(* IEC 61131-3 sources: LLM-CodeGen-TestGen/Tests/DEC_TO_HEX_2, 2 files *)

(* ---- DEC_TO_HEX_FullTest.st ---- *)
FUNCTION BIT_OF_DWORD : BOOL
  VAR_INPUT
    IN : DWORD;
    N : INT;
  END_VAR

  BIT_OF_DWORD := (SHR(in,N) AND 16#00000001) > 0;
  (* from OSCAT library; www.oscat.de  *)
END_FUNCTION

FUNCTION SIGN_R : BOOL
  VAR_INPUT
    IN : REAL;
  END_VAR

  SIGN_R := in < 0.0;
  (* from OSCAT library; www.oscat.de  *)
END_FUNCTION

FUNCTION FLOOR : INT
  VAR_INPUT
    x : REAL;
  END_VAR

  FLOOR := REAL_TO_INT(X);
  IF INT_TO_REAL(FLOOR) > X THEN
  	floor := floor - 1;
  END_IF;
  (* from OSCAT library; www.oscat.de  *)
END_FUNCTION

FUNCTION FLOOR2 : DINT
  VAR_INPUT
    x : REAL;
  END_VAR

  FLOOR2 := REAL_TO_DINT(X);
  IF DINT_TO_REAL(FLOOR2) > X THEN
  	FLOOR2 := FLOOR2 - DINT#1;
  END_IF;
  (* from OSCAT library; www.oscat.de  *)
END_FUNCTION

FUNCTION MODR : REAL
  VAR_INPUT
    IN : REAL;
    DIVI : REAL;
  END_VAR

  IF divi = 0.0 THEN
  	MODR := 0.0;
  ELSE
  	MODR := in - DINT_TO_REAL(FLOOR2(in / divi)) * divi;
  END_IF;
  (* from OSCAT library; www.oscat.de  *)
  (* FC FLOOR2 required *)
END_FUNCTION

FUNCTION REVERSE : BYTE
  VAR_INPUT
    IN : BYTE;
  END_VAR

  reverse := SHL(in,7) OR SHR(in,7) OR (ROR(in,3) AND BYTE#2#01000100) OR (ROL(in,3) AND BYTE#2#00100010)
  	OR (SHL(in,1) AND BYTE#2#00010000) OR (SHR(in,1) AND BYTE#2#00001000);

  (* Fromm Oscat Library, www.oscat.de *)
END_FUNCTION

FUNCTION REFLECT : DWORD
  VAR_INPUT
    DI : DWORD;
    L : INT;
  END_VAR
  VAR
    i : INT;
    _d : DWORD;
  END_VAR

  _d := DI;
  FOR i := 1 TO L DO
  	REFLECT := SHL(REFLECT, 1) OR BOOL_TO_DWORD((_d AND DWORD#2#0000_0001) > DWORD#0); (* D.0 *)
  	_d := SHR(_d, 1);
  END_FOR;
  REFLECT := REFLECT OR SHL(_d, L);

  (* Fromm Oscat Library, www.oscat.de *)
END_FUNCTION

FUNCTION BIT_LOAD_B : BYTE
  VAR_INPUT
    IN : BYTE;
    VAL : BOOL;
    POS : INT;
  END_VAR

  IF VAL THEN
  	BIT_LOAD_B := in OR SHL(BYTE#1,pos);
  ELSE
  	BIT_LOAD_B := in AND (NOT SHL(BYTE#1,pos));
  END_IF;

  (*From OSCAT Library, www.oscat.de*)
END_FUNCTION

FUNCTION _BYTE_TO_INT : INT
  VAR_INPUT
    IN : BYTE;
  END_VAR

  _BYTE_TO_INT := USINT_TO_INT(BYTE_TO_USINT(IN));

  (*From OSCAT Library, www.oscat.de*)
END_FUNCTION

FUNCTION T_PLC_MS : UDINT
  VAR
    tx : UDINT;
  END_VAR
  VAR_INPUT
    debug : BOOL;
  END_VAR
  VAR
    N : INT := 0;
    offset : UDINT := 0;
    temp : DWORD := 1;
  END_VAR

  tx := 0;
  {extern unsigned long __tick;
  extern unsigned long long common_ticktime__;
  unsigned long long ticktime_ms = (common_ticktime__)/1000000;
  UDINT plc_time = (UDINT)(ticktime_ms * (unsigned long long)__tick);
  TX = plc_time}
  T_PLC_MS := tx;
  IF debug THEN
  	T_PLC_MS := (DWORD_TO_UDINT(SHL(UDINT_TO_DWORD(T_PLC_MS),N) OR SHL(temp,N))-1) + OFFSET;
  END_IF;

  IF debug THEN
  	T_PLC_MS := (DWORD_TO_UDINT(SHL(UDINT_TO_DWORD(T_PLC_MS),N) OR SHL(temp,N))-1) + OFFSET;
  END_IF;

  (* Original Code:
  tx := TIME();
  T_PLC_MS := TIME_TO_DWORD(Tx);
  IF debug THEN
  	T_PLC_MS := (SHL(T_PLC_MS,N) OR SHL(DWORD#1,N)-1) + OFFSET;
  END_IF;
  *)

  (* From OSCAT library, www.oscat.de

  this is a temporary T_PLC_MS FB until OpenPLC gets it´s own time() functionality *)

  (* PLC_TIME and Global variables PLC_SCAN_CYCL and PLC_CYCL_TIME required *)
END_FUNCTION

FUNCTION T_PLC_US : UDINT
  VAR
    tx : UDINT;
  END_VAR
  VAR_INPUT
    debug : BOOL;
  END_VAR
  VAR
    N : INT := 0;
    offset : UDINT := 0;
    temp : DWORD := 1;
  END_VAR

  T_PLC_US := tx*1000;
  IF debug THEN
  	T_PLC_US := (DWORD_TO_UDINT(SHL(UDINT_TO_DWORD(T_PLC_US),N) OR SHL(temp,N))-1) + OFFSET;
  END_IF;

  (* Original Code:
  tx := TIME();
  T_PLC_US := TIME_TO_DWORD(Tx)*1000;
  IF debug THEN
  	T_PLC_US := (SHL(T_PLC_US,N) OR SHL(DWORD#1,N)-1) + OFFSET;
  END_IF;
  *)

  (* From OSCAT library, www.oscat.de

  this is a temporary T_PLC_US FB until OpenPLC gets it´s own time() functionality *)

  (* PLC_TIME and Global variables PLC_SCAN_CYCL and PLC_CYCL_TIME required *)
END_FUNCTION

FUNCTION_BLOCK FT_DERIV
  VAR_INPUT
    IN : REAL;
    K : REAL := 1.0;
    RUN : BOOL := TRUE;
  END_VAR
  VAR_OUTPUT
    OUT : REAL;
  END_VAR
  VAR
    old : REAL;
    tx : UDINT;
    last : UDINT;
    init : BOOL;
    tc : REAL;
  END_VAR

  tx:= T_PLC_US(en:=true);
  tc := UDINT_TO_REAL(tx - last);

  (* init on firsat startup *)
  IF NOT init THEN
  	init := TRUE;
  	old := in;
  ELSIF run AND tc > 0.0 THEN
  	out := (in - old) / tc * 1000000.0 * K;
  	old := in;
  ELSE
  	out := 0.0;
  END_IF;

  last := tx;

  (* From OSCAT Library, www.oscat.de *)
  (* T_PLC_US, required *)
END_FUNCTION_BLOCK

FUNCTION_BLOCK FT_PIWL
  VAR_INPUT
    IN : REAL;
    KP : REAL := 1.0;
    KI : REAL := 1.0;
    LIM_L : REAL := -1.0E38;
    LIM_H : REAL := 1.0E38;
    RST : BOOL;
  END_VAR
  VAR_OUTPUT
    Y : REAL;
    LIM : BOOL;
  END_VAR
  VAR
    init : BOOL;
    tx : UDINT;
    tc : REAL;
    t_last : UDINT;
    in_last : REAL;
    i : REAL;
    p : REAL;
  END_VAR

  IF NOT init OR RST THEN
  	init := TRUE;
  	in_last := in;
  		t_last := T_PLC_US(en:=true);
  	i := 0.0;
  	tc := 0.0;
  ELSE
  	(* read last cycle time in Microseconds *)
  		tx := T_PLC_US(en:=true);
  	tc := UDINT_TO_REAL(tx - t_last);
  	t_last := tx;

  	(* calculate proportional part *)
  	p := KP * IN;

  	(* run integrator *)
  	i := (IN + in_last) * 5.0E-7 * KI * tc + i;
  	in_last := IN;

  	(* calculate output Y *)
  	Y := p + i;

  	(* check output for limits *)
  	IF Y >= LIM_H THEN
  		Y := LIM_H;
  		IF ki <> 0.0 THEN
  			i := LIM_H - p;
  		ELSE
  			i := 0.0;
  		END_IF;
  		LIM := TRUE;
  	ELSIF Y <= LIM_L THEN
  		Y := LIM_L;
  		IF ki <> 0.0 THEN
  			i := LIM_L - p;
  		ELSE
  			i := 0.0;
  		END_IF;
  		LIM := TRUE;
  	ELSE
  		LIM := FALSE;
  	END_IF;
  END_IF;

  (* From OSCAT Library, www.oscat.de *)
  (* T_PLC_US required *)
END_FUNCTION_BLOCK

FUNCTION_BLOCK INTEGRATE
  VAR_INPUT
    _E : BOOL := TRUE;
    X : REAL;
    K : REAL := 1.0;
  END_VAR
  VAR_IN_OUT
    Y : REAL;
  END_VAR
  VAR
    x_last : REAL;
    init : BOOL;
    last : UDINT;
    tx : UDINT;
  END_VAR

  tx:= T_PLC_MS(en:=true);

  IF NOT init THEN
  	init := TRUE;
  	X_last := X;
  ELSIF _E THEN
  	Y := (X + X_LAST) * 0.5E-3 * UDINT_TO_REAL(tx-last) * K + Y;
  	X_last := X;
  END_IF;
  last := tx;

  (* From OSCAT Library, www.oscat.de *)
  (* T_PLC_MS required *)
END_FUNCTION_BLOCK

FUNCTION_BLOCK DEC_TO_HEX
  VAR_INPUT
    DecimalValue : DINT;
  END_VAR
  VAR_OUTPUT
    HexString : STRING;
  END_VAR
  VAR
    i : INT;
    hexDigits : ARRAY [0..15] OF STRING := ['0', '1', '2', '3', '4', '5', '6', '7', '8', '9', 'A', 'B', 'C', 'D', 'E', 'F'];
    digitIndex : INT;
    hexDigit : STRING;
    significantDigitFound : BOOL := FALSE;
    digitValue : DINT;
    powerOfInteger : DINT;
  END_VAR

  HexString := '';

  IF DecimalValue = 0 THEN
      HexString := '0';
      RETURN;
  END_IF;

  significantDigitFound := FALSE;

  FOR digitIndex := 0 TO 7 DO

      powerOfInteger:=1;
      FOR i := 1 TO 7 - digitIndex DO
        powerOfInteger := powerOfInteger * 16;
      END_FOR;

      digitValue := DIV(DecimalValue, powerOfInteger) MOD 16;
      hexDigit := hexDigits[digitValue];

      IF hexDigit <> '0' OR significantDigitFound OR (7 - digitIndex) = 0 THEN
          significantDigitFound := TRUE;
          HexString := CONCAT(HexString, hexDigit);
      END_IF;

  END_FOR;
END_FUNCTION_BLOCK

FUNCTION_BLOCK FB_TEST_0
  VAR_OUTPUT
    Finished : BOOL;
    Failed : BOOL;
  END_VAR
  VAR
    TestBlock : DEC_TO_HEX;
    TestState : INT;
    Timer : TON;
  END_VAR

  Timer(IN:=TRUE, PT:= T#0s); (* placeholder for later usage *)

  CASE testState OF
    0:
      IF (Timer.Q) THEN
        TestBlock(DecimalValue := 0);
        TestState:=TestState+1;
      END_IF;
      Timer(IN:=TRUE, PT:=T#0s);
    1:
      IF (Timer.Q) THEN
      {printf("0,0: TestBlock.HexString = '0'  actual=%s\n", (char*)&__GET_VAR(data__->TESTBLOCK.HEXSTRING,).body);}
        IF NOT(TestBlock.HexString = '0') THEN Failed := TRUE; END_IF;
      END_IF;
      Finished:=TRUE;
  END_CASE;
END_FUNCTION_BLOCK

FUNCTION_BLOCK FB_TEST_1
  VAR_OUTPUT
    Finished : BOOL;
    Failed : BOOL;
  END_VAR
  VAR
    TestBlock : DEC_TO_HEX;
    TestState : INT;
    Timer : TON;
  END_VAR

  Timer(IN:=TRUE, PT:= T#0s); (* placeholder for later usage *)

  CASE testState OF
    0:
      IF (Timer.Q) THEN
        TestBlock(DecimalValue := 1);
        TestState:=TestState+1;
      END_IF;
      Timer(IN:=TRUE, PT:=T#0s);
    1:
      IF (Timer.Q) THEN
      {printf("1,0: TestBlock.HexString = '1'  actual=%s\n", (char*)&__GET_VAR(data__->TESTBLOCK.HEXSTRING,).body);}
        IF NOT(TestBlock.HexString = '1') THEN Failed := TRUE; END_IF;
      END_IF;
      Finished:=TRUE;
  END_CASE;
END_FUNCTION_BLOCK

FUNCTION_BLOCK FB_TEST_2
  VAR_OUTPUT
    Finished : BOOL;
    Failed : BOOL;
  END_VAR
  VAR
    TestBlock : DEC_TO_HEX;
    TestState : INT;
    Timer : TON;
  END_VAR

  Timer(IN:=TRUE, PT:= T#0s); (* placeholder for later usage *)

  CASE testState OF
    0:
      IF (Timer.Q) THEN
        TestBlock(DecimalValue := 10);
        TestState:=TestState+1;
      END_IF;
      Timer(IN:=TRUE, PT:=T#0s);
    1:
      IF (Timer.Q) THEN
      {printf("2,0: TestBlock.HexString = 'A'  actual=%s\n", (char*)&__GET_VAR(data__->TESTBLOCK.HEXSTRING,).body);}
        IF NOT(TestBlock.HexString = 'A') THEN Failed := TRUE; END_IF;
      END_IF;
      Finished:=TRUE;
  END_CASE;
END_FUNCTION_BLOCK

FUNCTION_BLOCK FB_TEST_3
  VAR_OUTPUT
    Finished : BOOL;
    Failed : BOOL;
  END_VAR
  VAR
    TestBlock : DEC_TO_HEX;
    TestState : INT;
    Timer : TON;
  END_VAR

  Timer(IN:=TRUE, PT:= T#0s); (* placeholder for later usage *)

  CASE testState OF
    0:
      IF (Timer.Q) THEN
        TestBlock(DecimalValue := 15);
        TestState:=TestState+1;
      END_IF;
      Timer(IN:=TRUE, PT:=T#0s);
    1:
      IF (Timer.Q) THEN
      {printf("3,0: TestBlock.HexString = 'F'  actual=%s\n", (char*)&__GET_VAR(data__->TESTBLOCK.HEXSTRING,).body);}
        IF NOT(TestBlock.HexString = 'F') THEN Failed := TRUE; END_IF;
      END_IF;
      Finished:=TRUE;
  END_CASE;
END_FUNCTION_BLOCK

FUNCTION_BLOCK FB_TEST_4
  VAR_OUTPUT
    Finished : BOOL;
    Failed : BOOL;
  END_VAR
  VAR
    TestBlock : DEC_TO_HEX;
    TestState : INT;
    Timer : TON;
  END_VAR

  Timer(IN:=TRUE, PT:= T#0s); (* placeholder for later usage *)

  CASE testState OF
    0:
      IF (Timer.Q) THEN
        TestBlock(DecimalValue := 16);
        TestState:=TestState+1;
      END_IF;
      Timer(IN:=TRUE, PT:=T#0s);
    1:
      IF (Timer.Q) THEN
      {printf("4,0: TestBlock.HexString = '10'  actual=%s\n", (char*)&__GET_VAR(data__->TESTBLOCK.HEXSTRING,).body);}
        IF NOT(TestBlock.HexString = '10') THEN Failed := TRUE; END_IF;
      END_IF;
      Finished:=TRUE;
  END_CASE;
END_FUNCTION_BLOCK

FUNCTION_BLOCK FB_TEST_5
  VAR_OUTPUT
    Finished : BOOL;
    Failed : BOOL;
  END_VAR
  VAR
    TestBlock : DEC_TO_HEX;
    TestState : INT;
    Timer : TON;
  END_VAR

  Timer(IN:=TRUE, PT:= T#0s); (* placeholder for later usage *)

  CASE testState OF
    0:
      IF (Timer.Q) THEN
        TestBlock(DecimalValue := 255);
        TestState:=TestState+1;
      END_IF;
      Timer(IN:=TRUE, PT:=T#0s);
    1:
      IF (Timer.Q) THEN
      {printf("5,0: TestBlock.HexString = 'FF'  actual=%s\n", (char*)&__GET_VAR(data__->TESTBLOCK.HEXSTRING,).body);}
        IF NOT(TestBlock.HexString = 'FF') THEN Failed := TRUE; END_IF;
      END_IF;
      Finished:=TRUE;
  END_CASE;
END_FUNCTION_BLOCK

FUNCTION_BLOCK FB_TEST_6
  VAR_OUTPUT
    Finished : BOOL;
    Failed : BOOL;
  END_VAR
  VAR
    TestBlock : DEC_TO_HEX;
    TestState : INT;
    Timer : TON;
  END_VAR

  Timer(IN:=TRUE, PT:= T#0s); (* placeholder for later usage *)

  CASE testState OF
    0:
      IF (Timer.Q) THEN
        TestBlock(DecimalValue := 4095);
        TestState:=TestState+1;
      END_IF;
      Timer(IN:=TRUE, PT:=T#0s);
    1:
      IF (Timer.Q) THEN
      {printf("6,0: TestBlock.HexString = 'FFF'  actual=%s\n", (char*)&__GET_VAR(data__->TESTBLOCK.HEXSTRING,).body);}
        IF NOT(TestBlock.HexString = 'FFF') THEN Failed := TRUE; END_IF;
      END_IF;
      Finished:=TRUE;
  END_CASE;
END_FUNCTION_BLOCK

FUNCTION_BLOCK FB_TEST_7
  VAR_OUTPUT
    Finished : BOOL;
    Failed : BOOL;
  END_VAR
  VAR
    TestBlock : DEC_TO_HEX;
    TestState : INT;
    Timer : TON;
  END_VAR

  Timer(IN:=TRUE, PT:= T#0s); (* placeholder for later usage *)

  CASE testState OF
    0:
      IF (Timer.Q) THEN
        TestBlock(DecimalValue := 32767);
        TestState:=TestState+1;
      END_IF;
      Timer(IN:=TRUE, PT:=T#0s);
    1:
      IF (Timer.Q) THEN
      {printf("7,0: TestBlock.HexString = '7FFF'  actual=%s\n", (char*)&__GET_VAR(data__->TESTBLOCK.HEXSTRING,).body);}
        IF NOT(TestBlock.HexString = '7FFF') THEN Failed := TRUE; END_IF;
      END_IF;
      Finished:=TRUE;
  END_CASE;
END_FUNCTION_BLOCK

FUNCTION_BLOCK FB_TEST_8
  VAR_OUTPUT
    Finished : BOOL;
    Failed : BOOL;
  END_VAR
  VAR
    TestBlock : DEC_TO_HEX;
    TestState : INT;
    Timer : TON;
  END_VAR

  Timer(IN:=TRUE, PT:= T#0s); (* placeholder for later usage *)

  CASE testState OF
    0:
      IF (Timer.Q) THEN
        TestBlock(DecimalValue := 32768);
        TestState:=TestState+1;
      END_IF;
      Timer(IN:=TRUE, PT:=T#0s);
    1:
      IF (Timer.Q) THEN
      {printf("8,0: TestBlock.HexString = '8000'  actual=%s\n", (char*)&__GET_VAR(data__->TESTBLOCK.HEXSTRING,).body);}
        IF NOT(TestBlock.HexString = '8000') THEN Failed := TRUE; END_IF;
      END_IF;
      Finished:=TRUE;
  END_CASE;
END_FUNCTION_BLOCK

FUNCTION_BLOCK FB_TEST_9
  VAR_OUTPUT
    Finished : BOOL;
    Failed : BOOL;
  END_VAR
  VAR
    TestBlock : DEC_TO_HEX;
    TestState : INT;
    Timer : TON;
  END_VAR

  Timer(IN:=TRUE, PT:= T#0s); (* placeholder for later usage *)

  CASE testState OF
    0:
      IF (Timer.Q) THEN
        TestBlock(DecimalValue := 65535);
        TestState:=TestState+1;
      END_IF;
      Timer(IN:=TRUE, PT:=T#0s);
    1:
      IF (Timer.Q) THEN
      {printf("9,0: TestBlock.HexString = 'FFFF'  actual=%s\n", (char*)&__GET_VAR(data__->TESTBLOCK.HEXSTRING,).body);}
        IF NOT(TestBlock.HexString = 'FFFF') THEN Failed := TRUE; END_IF;
      END_IF;
      Finished:=TRUE;
  END_CASE;
END_FUNCTION_BLOCK

FUNCTION_BLOCK FB_TEST_10
  VAR_OUTPUT
    Finished : BOOL;
    Failed : BOOL;
  END_VAR
  VAR
    TestBlock : DEC_TO_HEX;
    TestState : INT;
    Timer : TON;
  END_VAR

  Timer(IN:=TRUE, PT:= T#0s); (* placeholder for later usage *)

  CASE testState OF
    0:
      IF (Timer.Q) THEN
        TestBlock(DecimalValue := -32768);
        TestState:=TestState+1;
      END_IF;
      Timer(IN:=TRUE, PT:=T#0s);
    1:
      IF (Timer.Q) THEN
      {printf("10,0: TestBlock.HexString = '8000'  actual=%s\n", (char*)&__GET_VAR(data__->TESTBLOCK.HEXSTRING,).body);}
        IF NOT(TestBlock.HexString = '8000') THEN Failed := TRUE; END_IF;
      END_IF;
      Finished:=TRUE;
  END_CASE;
END_FUNCTION_BLOCK

FUNCTION_BLOCK FB_TEST_11
  VAR_OUTPUT
    Finished : BOOL;
    Failed : BOOL;
  END_VAR
  VAR
    TestBlock : DEC_TO_HEX;
    TestState : INT;
    Timer : TON;
  END_VAR

  Timer(IN:=TRUE, PT:= T#0s); (* placeholder for later usage *)

  CASE testState OF
    0:
      IF (Timer.Q) THEN
        TestBlock(DecimalValue := -1);
        TestState:=TestState+1;
      END_IF;
      Timer(IN:=TRUE, PT:=T#0s);
    1:
      IF (Timer.Q) THEN
      {printf("11,0: TestBlock.HexString = 'FFFFFFFF'  actual=%s\n", (char*)&__GET_VAR(data__->TESTBLOCK.HEXSTRING,).body);}
        IF NOT(TestBlock.HexString = 'FFFFFFFF') THEN Failed := TRUE; END_IF;
      END_IF;
      Finished:=TRUE;
  END_CASE;
END_FUNCTION_BLOCK

FUNCTION_BLOCK FB_TEST_12
  VAR_OUTPUT
    Finished : BOOL;
    Failed : BOOL;
  END_VAR
  VAR
    TestBlock : DEC_TO_HEX;
    TestState : INT;
    Timer : TON;
  END_VAR

  Timer(IN:=TRUE, PT:= T#0s); (* placeholder for later usage *)

  CASE testState OF
    0:
      IF (Timer.Q) THEN
        TestBlock(DecimalValue := -16);
        TestState:=TestState+1;
      END_IF;
      Timer(IN:=TRUE, PT:=T#0s);
    1:
      IF (Timer.Q) THEN
      {printf("12,0: TestBlock.HexString = 'FFFFFFF0'  actual=%s\n", (char*)&__GET_VAR(data__->TESTBLOCK.HEXSTRING,).body);}
        IF NOT(TestBlock.HexString = 'FFFFFFF0') THEN Failed := TRUE; END_IF;
      END_IF;
      Finished:=TRUE;
  END_CASE;
END_FUNCTION_BLOCK

FUNCTION_BLOCK FB_TEST_13
  VAR_OUTPUT
    Finished : BOOL;
    Failed : BOOL;
  END_VAR
  VAR
    TestBlock : DEC_TO_HEX;
    TestState : INT;
    Timer : TON;
  END_VAR

  Timer(IN:=TRUE, PT:= T#0s); (* placeholder for later usage *)

  CASE testState OF
    0:
      IF (Timer.Q) THEN
        TestBlock(DecimalValue := -255);
        TestState:=TestState+1;
      END_IF;
      Timer(IN:=TRUE, PT:=T#0s);
    1:
      IF (Timer.Q) THEN
      {printf("13,0: TestBlock.HexString = 'FFFFFF01'  actual=%s\n", (char*)&__GET_VAR(data__->TESTBLOCK.HEXSTRING,).body);}
        IF NOT(TestBlock.HexString = 'FFFFFF01') THEN Failed := TRUE; END_IF;
      END_IF;
      Finished:=TRUE;
  END_CASE;
END_FUNCTION_BLOCK

FUNCTION_BLOCK FB_TEST_14
  VAR_OUTPUT
    Finished : BOOL;
    Failed : BOOL;
  END_VAR
  VAR
    TestBlock : DEC_TO_HEX;
    TestState : INT;
    Timer : TON;
  END_VAR

  Timer(IN:=TRUE, PT:= T#0s); (* placeholder for later usage *)

  CASE testState OF
    0:
      IF (Timer.Q) THEN
        TestBlock(DecimalValue := -4095);
        TestState:=TestState+1;
      END_IF;
      Timer(IN:=TRUE, PT:=T#0s);
    1:
      IF (Timer.Q) THEN
      {printf("14,0: TestBlock.HexString = 'FFFFF001'  actual=%s\n", (char*)&__GET_VAR(data__->TESTBLOCK.HEXSTRING,).body);}
        IF NOT(TestBlock.HexString = 'FFFFF001') THEN Failed := TRUE; END_IF;
      END_IF;
      Finished:=TRUE;
  END_CASE;
END_FUNCTION_BLOCK

FUNCTION_BLOCK FB_TEST_15
  VAR_OUTPUT
    Finished : BOOL;
    Failed : BOOL;
  END_VAR
  VAR
    TestBlock : DEC_TO_HEX;
    TestState : INT;
    Timer : TON;
  END_VAR

  Timer(IN:=TRUE, PT:= T#0s); (* placeholder for later usage *)

  CASE testState OF
    0:
      IF (Timer.Q) THEN
        TestBlock(DecimalValue := -32767);
        TestState:=TestState+1;
      END_IF;
      Timer(IN:=TRUE, PT:=T#0s);
    1:
      IF (Timer.Q) THEN
      {printf("15,0: TestBlock.HexString = 'FFFF8001'  actual=%s\n", (char*)&__GET_VAR(data__->TESTBLOCK.HEXSTRING,).body);}
        IF NOT(TestBlock.HexString = 'FFFF8001') THEN Failed := TRUE; END_IF;
      END_IF;
      Finished:=TRUE;
  END_CASE;
END_FUNCTION_BLOCK

FUNCTION_BLOCK FB_TEST_16
  VAR_OUTPUT
    Finished : BOOL;
    Failed : BOOL;
  END_VAR
  VAR
    TestBlock : DEC_TO_HEX;
    TestState : INT;
    Timer : TON;
  END_VAR

  Timer(IN:=TRUE, PT:= T#0s); (* placeholder for later usage *)

  CASE testState OF
    0:
      IF (Timer.Q) THEN
        TestBlock(DecimalValue := -32768);
        TestState:=TestState+1;
      END_IF;
      Timer(IN:=TRUE, PT:=T#0s);
    1:
      IF (Timer.Q) THEN
      {printf("16,0: TestBlock.HexString = 'FFFF8000'  actual=%s\n", (char*)&__GET_VAR(data__->TESTBLOCK.HEXSTRING,).body);}
        IF NOT(TestBlock.HexString = 'FFFF8000') THEN Failed := TRUE; END_IF;
      END_IF;
      Finished:=TRUE;
  END_CASE;
END_FUNCTION_BLOCK

FUNCTION_BLOCK FB_TEST_17
  VAR_OUTPUT
    Finished : BOOL;
    Failed : BOOL;
  END_VAR
  VAR
    TestBlock : DEC_TO_HEX;
    TestState : INT;
    Timer : TON;
  END_VAR

  Timer(IN:=TRUE, PT:= T#0s); (* placeholder for later usage *)

  CASE testState OF
    0:
      IF (Timer.Q) THEN
        TestBlock(DecimalValue := -65535);
        TestState:=TestState+1;
      END_IF;
      Timer(IN:=TRUE, PT:=T#0s);
    1:
      IF (Timer.Q) THEN
      {printf("17,0: TestBlock.HexString = 'FFFF0001'  actual=%s\n", (char*)&__GET_VAR(data__->TESTBLOCK.HEXSTRING,).body);}
        IF NOT(TestBlock.HexString = 'FFFF0001') THEN Failed := TRUE; END_IF;
      END_IF;
      Finished:=TRUE;
  END_CASE;
END_FUNCTION_BLOCK

PROGRAM TestRunnerProgram
VAR
  testResult AT %QX0.0 : BOOL := FALSE;
END_VAR
VAR
  totalTests AT %QW0 : INT := 0;
  passedTests AT %QW1 : INT := 0;
END_VAR
VAR
  i: INT := 0;
  testOutcomeArray : ARRAY [0..17] OF BOOL;
  Test_0: FB_TEST_0;
  Test_1: FB_TEST_1;
  Test_2: FB_TEST_2;
  Test_3: FB_TEST_3;
  Test_4: FB_TEST_4;
  Test_5: FB_TEST_5;
  Test_6: FB_TEST_6;
  Test_7: FB_TEST_7;
  Test_8: FB_TEST_8;
  Test_9: FB_TEST_9;
  Test_10: FB_TEST_10;
  Test_11: FB_TEST_11;
  Test_12: FB_TEST_12;
  Test_13: FB_TEST_13;
  Test_14: FB_TEST_14;
  Test_15: FB_TEST_15;
  Test_16: FB_TEST_16;
  Test_17: FB_TEST_17;
END_VAR

  IF NOT Test_0.Finished AND NOT Test_0.FAILED THEN totalTests := totalTests + 1; Test_0(); END_IF;
  IF Test_0.Finished THEN testOutcomeArray[0] := TRUE; END_IF;
  IF NOT Test_1.Finished AND NOT Test_1.FAILED THEN totalTests := totalTests + 1; Test_1(); END_IF;
  IF Test_1.Finished THEN testOutcomeArray[1] := TRUE; END_IF;
  IF NOT Test_2.Finished AND NOT Test_2.FAILED THEN totalTests := totalTests + 1; Test_2(); END_IF;
  IF Test_2.Finished THEN testOutcomeArray[2] := TRUE; END_IF;
  IF NOT Test_3.Finished AND NOT Test_3.FAILED THEN totalTests := totalTests + 1; Test_3(); END_IF;
  IF Test_3.Finished THEN testOutcomeArray[3] := TRUE; END_IF;
  IF NOT Test_4.Finished AND NOT Test_4.FAILED THEN totalTests := totalTests + 1; Test_4(); END_IF;
  IF Test_4.Finished THEN testOutcomeArray[4] := TRUE; END_IF;
  IF NOT Test_5.Finished AND NOT Test_5.FAILED THEN totalTests := totalTests + 1; Test_5(); END_IF;
  IF Test_5.Finished THEN testOutcomeArray[5] := TRUE; END_IF;
  IF NOT Test_6.Finished AND NOT Test_6.FAILED THEN totalTests := totalTests + 1; Test_6(); END_IF;
  IF Test_6.Finished THEN testOutcomeArray[6] := TRUE; END_IF;
  IF NOT Test_7.Finished AND NOT Test_7.FAILED THEN totalTests := totalTests + 1; Test_7(); END_IF;
  IF Test_7.Finished THEN testOutcomeArray[7] := TRUE; END_IF;
  IF NOT Test_8.Finished AND NOT Test_8.FAILED THEN totalTests := totalTests + 1; Test_8(); END_IF;
  IF Test_8.Finished THEN testOutcomeArray[8] := TRUE; END_IF;
  IF NOT Test_9.Finished AND NOT Test_9.FAILED THEN totalTests := totalTests + 1; Test_9(); END_IF;
  IF Test_9.Finished THEN testOutcomeArray[9] := TRUE; END_IF;
  IF NOT Test_10.Finished AND NOT Test_10.FAILED THEN totalTests := totalTests + 1; Test_10(); END_IF;
  IF Test_10.Finished THEN testOutcomeArray[10] := TRUE; END_IF;
  IF NOT Test_11.Finished AND NOT Test_11.FAILED THEN totalTests := totalTests + 1; Test_11(); END_IF;
  IF Test_11.Finished THEN testOutcomeArray[11] := TRUE; END_IF;
  IF NOT Test_12.Finished AND NOT Test_12.FAILED THEN totalTests := totalTests + 1; Test_12(); END_IF;
  IF Test_12.Finished THEN testOutcomeArray[12] := TRUE; END_IF;
  IF NOT Test_13.Finished AND NOT Test_13.FAILED THEN totalTests := totalTests + 1; Test_13(); END_IF;
  IF Test_13.Finished THEN testOutcomeArray[13] := TRUE; END_IF;
  IF NOT Test_14.Finished AND NOT Test_14.FAILED THEN totalTests := totalTests + 1; Test_14(); END_IF;
  IF Test_14.Finished THEN testOutcomeArray[14] := TRUE; END_IF;
  IF NOT Test_15.Finished AND NOT Test_15.FAILED THEN totalTests := totalTests + 1; Test_15(); END_IF;
  IF Test_15.Finished THEN testOutcomeArray[15] := TRUE; END_IF;
  IF NOT Test_16.Finished AND NOT Test_16.FAILED THEN totalTests := totalTests + 1; Test_16(); END_IF;
  IF Test_16.Finished THEN testOutcomeArray[16] := TRUE; END_IF;
  IF NOT Test_17.Finished AND NOT Test_17.FAILED THEN totalTests := totalTests + 1; Test_17(); END_IF;
  IF Test_17.Finished THEN testOutcomeArray[17] := TRUE; END_IF;

  passedTests := 0;
  FOR i:=0 TO 17 DO
    IF testOutcomeArray[i]=TRUE THEN passedTests := passedTests+1; END_IF;
  END_FOR;
END_PROGRAM

CONFIGURATION Config0

  RESOURCE Res0 ON PLC
    TASK task0(INTERVAL := T#100ms,PRIORITY := 0);
    PROGRAM instance0 WITH task0 : TestRunnerProgram;
  END_RESOURCE
END_CONFIGURATION

(* ---- DEC_TO_HEX_TestCases.st ---- *)
FUNCTION_BLOCK FB_TEST_0
  VAR_OUTPUT
    Finished : BOOL;
    Failed : BOOL;
  END_VAR
  VAR
    TestBlock : DEC_TO_HEX;
    TestState : INT;
    Timer : TON;
  END_VAR

  Timer(IN:=TRUE, PT:= T#0s); (* placeholder for later usage *)

  CASE testState OF
    0:
      IF (Timer.Q) THEN
        TestBlock(DecimalValue := 0);
        TestState:=TestState+1;
      END_IF;
      Timer(IN:=TRUE, PT:=T#0s);
    1:
      IF (Timer.Q) THEN
      {printf("0,0: TestBlock.HexString = '0'  actual=%lf\n", (double)__GET_VAR(data__->TESTBLOCK.HEXSTRING,));}
        IF NOT(TestBlock.HexString = '0') THEN Failed := TRUE; END_IF;
      END_IF;
      Finished:=TRUE;
  END_CASE;
END_FUNCTION_BLOCK

FUNCTION_BLOCK FB_TEST_1
  VAR_OUTPUT
    Finished : BOOL;
    Failed : BOOL;
  END_VAR
  VAR
    TestBlock : DEC_TO_HEX;
    TestState : INT;
    Timer : TON;
  END_VAR

  Timer(IN:=TRUE, PT:= T#0s); (* placeholder for later usage *)

  CASE testState OF
    0:
      IF (Timer.Q) THEN
        TestBlock(DecimalValue := 1);
        TestState:=TestState+1;
      END_IF;
      Timer(IN:=TRUE, PT:=T#0s);
    1:
      IF (Timer.Q) THEN
      {printf("1,0: TestBlock.HexString = '1'  actual=%lf\n", (double)__GET_VAR(data__->TESTBLOCK.HEXSTRING,));}
        IF NOT(TestBlock.HexString = '1') THEN Failed := TRUE; END_IF;
      END_IF;
      Finished:=TRUE;
  END_CASE;
END_FUNCTION_BLOCK

FUNCTION_BLOCK FB_TEST_2
  VAR_OUTPUT
    Finished : BOOL;
    Failed : BOOL;
  END_VAR
  VAR
    TestBlock : DEC_TO_HEX;
    TestState : INT;
    Timer : TON;
  END_VAR

  Timer(IN:=TRUE, PT:= T#0s); (* placeholder for later usage *)

  CASE testState OF
    0:
      IF (Timer.Q) THEN
        TestBlock(DecimalValue := 10);
        TestState:=TestState+1;
      END_IF;
      Timer(IN:=TRUE, PT:=T#0s);
    1:
      IF (Timer.Q) THEN
      {printf("2,0: TestBlock.HexString = 'A'  actual=%lf\n", (double)__GET_VAR(data__->TESTBLOCK.HEXSTRING,));}
        IF NOT(TestBlock.HexString = 'A') THEN Failed := TRUE; END_IF;
      END_IF;
      Finished:=TRUE;
  END_CASE;
END_FUNCTION_BLOCK

FUNCTION_BLOCK FB_TEST_3
  VAR_OUTPUT
    Finished : BOOL;
    Failed : BOOL;
  END_VAR
  VAR
    TestBlock : DEC_TO_HEX;
    TestState : INT;
    Timer : TON;
  END_VAR

  Timer(IN:=TRUE, PT:= T#0s); (* placeholder for later usage *)

  CASE testState OF
    0:
      IF (Timer.Q) THEN
        TestBlock(DecimalValue := 15);
        TestState:=TestState+1;
      END_IF;
      Timer(IN:=TRUE, PT:=T#0s);
    1:
      IF (Timer.Q) THEN
      {printf("3,0: TestBlock.HexString = 'F'  actual=%lf\n", (double)__GET_VAR(data__->TESTBLOCK.HEXSTRING,));}
        IF NOT(TestBlock.HexString = 'F') THEN Failed := TRUE; END_IF;
      END_IF;
      Finished:=TRUE;
  END_CASE;
END_FUNCTION_BLOCK

FUNCTION_BLOCK FB_TEST_4
  VAR_OUTPUT
    Finished : BOOL;
    Failed : BOOL;
  END_VAR
  VAR
    TestBlock : DEC_TO_HEX;
    TestState : INT;
    Timer : TON;
  END_VAR

  Timer(IN:=TRUE, PT:= T#0s); (* placeholder for later usage *)

  CASE testState OF
    0:
      IF (Timer.Q) THEN
        TestBlock(DecimalValue := 16);
        TestState:=TestState+1;
      END_IF;
      Timer(IN:=TRUE, PT:=T#0s);
    1:
      IF (Timer.Q) THEN
      {printf("4,0: TestBlock.HexString = '10'  actual=%lf\n", (double)__GET_VAR(data__->TESTBLOCK.HEXSTRING,));}
        IF NOT(TestBlock.HexString = '10') THEN Failed := TRUE; END_IF;
      END_IF;
      Finished:=TRUE;
  END_CASE;
END_FUNCTION_BLOCK

FUNCTION_BLOCK FB_TEST_5
  VAR_OUTPUT
    Finished : BOOL;
    Failed : BOOL;
  END_VAR
  VAR
    TestBlock : DEC_TO_HEX;
    TestState : INT;
    Timer : TON;
  END_VAR

  Timer(IN:=TRUE, PT:= T#0s); (* placeholder for later usage *)

  CASE testState OF
    0:
      IF (Timer.Q) THEN
        TestBlock(DecimalValue := 255);
        TestState:=TestState+1;
      END_IF;
      Timer(IN:=TRUE, PT:=T#0s);
    1:
      IF (Timer.Q) THEN
      {printf("5,0: TestBlock.HexString = 'FF'  actual=%lf\n", (double)__GET_VAR(data__->TESTBLOCK.HEXSTRING,));}
        IF NOT(TestBlock.HexString = 'FF') THEN Failed := TRUE; END_IF;
      END_IF;
      Finished:=TRUE;
  END_CASE;
END_FUNCTION_BLOCK

FUNCTION_BLOCK FB_TEST_6
  VAR_OUTPUT
    Finished : BOOL;
    Failed : BOOL;
  END_VAR
  VAR
    TestBlock : DEC_TO_HEX;
    TestState : INT;
    Timer : TON;
  END_VAR

  Timer(IN:=TRUE, PT:= T#0s); (* placeholder for later usage *)

  CASE testState OF
    0:
      IF (Timer.Q) THEN
        TestBlock(DecimalValue := 4095);
        TestState:=TestState+1;
      END_IF;
      Timer(IN:=TRUE, PT:=T#0s);
    1:
      IF (Timer.Q) THEN
      {printf("6,0: TestBlock.HexString = 'FFF'  actual=%lf\n", (double)__GET_VAR(data__->TESTBLOCK.HEXSTRING,));}
        IF NOT(TestBlock.HexString = 'FFF') THEN Failed := TRUE; END_IF;
      END_IF;
      Finished:=TRUE;
  END_CASE;
END_FUNCTION_BLOCK

FUNCTION_BLOCK FB_TEST_7
  VAR_OUTPUT
    Finished : BOOL;
    Failed : BOOL;
  END_VAR
  VAR
    TestBlock : DEC_TO_HEX;
    TestState : INT;
    Timer : TON;
  END_VAR

  Timer(IN:=TRUE, PT:= T#0s); (* placeholder for later usage *)

  CASE testState OF
    0:
      IF (Timer.Q) THEN
        TestBlock(DecimalValue := 32767);
        TestState:=TestState+1;
      END_IF;
      Timer(IN:=TRUE, PT:=T#0s);
    1:
      IF (Timer.Q) THEN
      {printf("7,0: TestBlock.HexString = '7FFF'  actual=%lf\n", (double)__GET_VAR(data__->TESTBLOCK.HEXSTRING,));}
        IF NOT(TestBlock.HexString = '7FFF') THEN Failed := TRUE; END_IF;
      END_IF;
      Finished:=TRUE;
  END_CASE;
END_FUNCTION_BLOCK

FUNCTION_BLOCK FB_TEST_8
  VAR_OUTPUT
    Finished : BOOL;
    Failed : BOOL;
  END_VAR
  VAR
    TestBlock : DEC_TO_HEX;
    TestState : INT;
    Timer : TON;
  END_VAR

  Timer(IN:=TRUE, PT:= T#0s); (* placeholder for later usage *)

  CASE testState OF
    0:
      IF (Timer.Q) THEN
        TestBlock(DecimalValue := 32768);
        TestState:=TestState+1;
      END_IF;
      Timer(IN:=TRUE, PT:=T#0s);
    1:
      IF (Timer.Q) THEN
      {printf("8,0: TestBlock.HexString = '8000'  actual=%lf\n", (double)__GET_VAR(data__->TESTBLOCK.HEXSTRING,));}
        IF NOT(TestBlock.HexString = '8000') THEN Failed := TRUE; END_IF;
      END_IF;
      Finished:=TRUE;
  END_CASE;
END_FUNCTION_BLOCK

FUNCTION_BLOCK FB_TEST_9
  VAR_OUTPUT
    Finished : BOOL;
    Failed : BOOL;
  END_VAR
  VAR
    TestBlock : DEC_TO_HEX;
    TestState : INT;
    Timer : TON;
  END_VAR

  Timer(IN:=TRUE, PT:= T#0s); (* placeholder for later usage *)

  CASE testState OF
    0:
      IF (Timer.Q) THEN
        TestBlock(DecimalValue := 65535);
        TestState:=TestState+1;
      END_IF;
      Timer(IN:=TRUE, PT:=T#0s);
    1:
      IF (Timer.Q) THEN
      {printf("9,0: TestBlock.HexString = 'FFFF'  actual=%lf\n", (double)__GET_VAR(data__->TESTBLOCK.HEXSTRING,));}
        IF NOT(TestBlock.HexString = 'FFFF') THEN Failed := TRUE; END_IF;
      END_IF;
      Finished:=TRUE;
  END_CASE;
END_FUNCTION_BLOCK

FUNCTION_BLOCK FB_TEST_10
  VAR_OUTPUT
    Finished : BOOL;
    Failed : BOOL;
  END_VAR
  VAR
    TestBlock : DEC_TO_HEX;
    TestState : INT;
    Timer : TON;
  END_VAR

  Timer(IN:=TRUE, PT:= T#0s); (* placeholder for later usage *)

  CASE testState OF
    0:
      IF (Timer.Q) THEN
        TestBlock(DecimalValue := -32768);
        TestState:=TestState+1;
      END_IF;
      Timer(IN:=TRUE, PT:=T#0s);
    1:
      IF (Timer.Q) THEN
      {printf("10,0: TestBlock.HexString = '8000'  actual=%lf\n", (double)__GET_VAR(data__->TESTBLOCK.HEXSTRING,));}
        IF NOT(TestBlock.HexString = '8000') THEN Failed := TRUE; END_IF;
      END_IF;
      Finished:=TRUE;
  END_CASE;
END_FUNCTION_BLOCK

FUNCTION_BLOCK FB_TEST_11
  VAR_OUTPUT
    Finished : BOOL;
    Failed : BOOL;
  END_VAR
  VAR
    TestBlock : DEC_TO_HEX;
    TestState : INT;
    Timer : TON;
  END_VAR

  Timer(IN:=TRUE, PT:= T#0s); (* placeholder for later usage *)

  CASE testState OF
    0:
      IF (Timer.Q) THEN
        TestBlock(DecimalValue := -1);
        TestState:=TestState+1;
      END_IF;
      Timer(IN:=TRUE, PT:=T#0s);
    1:
      IF (Timer.Q) THEN
      {printf("11,0: TestBlock.HexString = 'FFFFFFFF'  actual=%lf\n", (double)__GET_VAR(data__->TESTBLOCK.HEXSTRING,));}
        IF NOT(TestBlock.HexString = 'FFFFFFFF') THEN Failed := TRUE; END_IF;
      END_IF;
      Finished:=TRUE;
  END_CASE;
END_FUNCTION_BLOCK

FUNCTION_BLOCK FB_TEST_12
  VAR_OUTPUT
    Finished : BOOL;
    Failed : BOOL;
  END_VAR
  VAR
    TestBlock : DEC_TO_HEX;
    TestState : INT;
    Timer : TON;
  END_VAR

  Timer(IN:=TRUE, PT:= T#0s); (* placeholder for later usage *)

  CASE testState OF
    0:
      IF (Timer.Q) THEN
        TestBlock(DecimalValue := -16);
        TestState:=TestState+1;
      END_IF;
      Timer(IN:=TRUE, PT:=T#0s);
    1:
      IF (Timer.Q) THEN
      {printf("12,0: TestBlock.HexString = 'FFFFFFF0'  actual=%lf\n", (double)__GET_VAR(data__->TESTBLOCK.HEXSTRING,));}
        IF NOT(TestBlock.HexString = 'FFFFFFF0') THEN Failed := TRUE; END_IF;
      END_IF;
      Finished:=TRUE;
  END_CASE;
END_FUNCTION_BLOCK

FUNCTION_BLOCK FB_TEST_13
  VAR_OUTPUT
    Finished : BOOL;
    Failed : BOOL;
  END_VAR
  VAR
    TestBlock : DEC_TO_HEX;
    TestState : INT;
    Timer : TON;
  END_VAR

  Timer(IN:=TRUE, PT:= T#0s); (* placeholder for later usage *)

  CASE testState OF
    0:
      IF (Timer.Q) THEN
        TestBlock(DecimalValue := -255);
        TestState:=TestState+1;
      END_IF;
      Timer(IN:=TRUE, PT:=T#0s);
    1:
      IF (Timer.Q) THEN
      {printf("13,0: TestBlock.HexString = 'FFFFFF01'  actual=%lf\n", (double)__GET_VAR(data__->TESTBLOCK.HEXSTRING,));}
        IF NOT(TestBlock.HexString = 'FFFFFF01') THEN Failed := TRUE; END_IF;
      END_IF;
      Finished:=TRUE;
  END_CASE;
END_FUNCTION_BLOCK

FUNCTION_BLOCK FB_TEST_14
  VAR_OUTPUT
    Finished : BOOL;
    Failed : BOOL;
  END_VAR
  VAR
    TestBlock : DEC_TO_HEX;
    TestState : INT;
    Timer : TON;
  END_VAR

  Timer(IN:=TRUE, PT:= T#0s); (* placeholder for later usage *)

  CASE testState OF
    0:
      IF (Timer.Q) THEN
        TestBlock(DecimalValue := -4095);
        TestState:=TestState+1;
      END_IF;
      Timer(IN:=TRUE, PT:=T#0s);
    1:
      IF (Timer.Q) THEN
      {printf("14,0: TestBlock.HexString = 'FFFFF001'  actual=%lf\n", (double)__GET_VAR(data__->TESTBLOCK.HEXSTRING,));}
        IF NOT(TestBlock.HexString = 'FFFFF001') THEN Failed := TRUE; END_IF;
      END_IF;
      Finished:=TRUE;
  END_CASE;
END_FUNCTION_BLOCK

FUNCTION_BLOCK FB_TEST_15
  VAR_OUTPUT
    Finished : BOOL;
    Failed : BOOL;
  END_VAR
  VAR
    TestBlock : DEC_TO_HEX;
    TestState : INT;
    Timer : TON;
  END_VAR

  Timer(IN:=TRUE, PT:= T#0s); (* placeholder for later usage *)

  CASE testState OF
    0:
      IF (Timer.Q) THEN
        TestBlock(DecimalValue := -32767);
        TestState:=TestState+1;
      END_IF;
      Timer(IN:=TRUE, PT:=T#0s);
    1:
      IF (Timer.Q) THEN
      {printf("15,0: TestBlock.HexString = 'FFFF8001'  actual=%lf\n", (double)__GET_VAR(data__->TESTBLOCK.HEXSTRING,));}
        IF NOT(TestBlock.HexString = 'FFFF8001') THEN Failed := TRUE; END_IF;
      END_IF;
      Finished:=TRUE;
  END_CASE;
END_FUNCTION_BLOCK

FUNCTION_BLOCK FB_TEST_16
  VAR_OUTPUT
    Finished : BOOL;
    Failed : BOOL;
  END_VAR
  VAR
    TestBlock : DEC_TO_HEX;
    TestState : INT;
    Timer : TON;
  END_VAR

  Timer(IN:=TRUE, PT:= T#0s); (* placeholder for later usage *)

  CASE testState OF
    0:
      IF (Timer.Q) THEN
        TestBlock(DecimalValue := -32768);
        TestState:=TestState+1;
      END_IF;
      Timer(IN:=TRUE, PT:=T#0s);
    1:
      IF (Timer.Q) THEN
      {printf("16,0: TestBlock.HexString = 'FFFF8000'  actual=%lf\n", (double)__GET_VAR(data__->TESTBLOCK.HEXSTRING,));}
        IF NOT(TestBlock.HexString = 'FFFF8000') THEN Failed := TRUE; END_IF;
      END_IF;
      Finished:=TRUE;
  END_CASE;
END_FUNCTION_BLOCK

FUNCTION_BLOCK FB_TEST_17
  VAR_OUTPUT
    Finished : BOOL;
    Failed : BOOL;
  END_VAR
  VAR
    TestBlock : DEC_TO_HEX;
    TestState : INT;
    Timer : TON;
  END_VAR

  Timer(IN:=TRUE, PT:= T#0s); (* placeholder for later usage *)

  CASE testState OF
    0:
      IF (Timer.Q) THEN
        TestBlock(DecimalValue := -65535);
        TestState:=TestState+1;
      END_IF;
      Timer(IN:=TRUE, PT:=T#0s);
    1:
      IF (Timer.Q) THEN
      {printf("17,0: TestBlock.HexString = 'FFFF0001'  actual=%lf\n", (double)__GET_VAR(data__->TESTBLOCK.HEXSTRING,));}
        IF NOT(TestBlock.HexString = 'FFFF0001') THEN Failed := TRUE; END_IF;
      END_IF;
      Finished:=TRUE;
  END_CASE;
END_FUNCTION_BLOCK

PROGRAM TestRunnerProgram
VAR
  testResult AT %QX0.0 : BOOL := FALSE;
END_VAR
VAR
  totalTests AT %QW0 : INT := 0;
  passedTests AT %QW1 : INT := 0;
END_VAR
VAR
  i: INT := 0;
  testOutcomeArray : ARRAY [0..17] OF BOOL;
  Test_0: FB_TEST_0;
  Test_1: FB_TEST_1;
  Test_2: FB_TEST_2;
  Test_3: FB_TEST_3;
  Test_4: FB_TEST_4;
  Test_5: FB_TEST_5;
  Test_6: FB_TEST_6;
  Test_7: FB_TEST_7;
  Test_8: FB_TEST_8;
  Test_9: FB_TEST_9;
  Test_10: FB_TEST_10;
  Test_11: FB_TEST_11;
  Test_12: FB_TEST_12;
  Test_13: FB_TEST_13;
  Test_14: FB_TEST_14;
  Test_15: FB_TEST_15;
  Test_16: FB_TEST_16;
  Test_17: FB_TEST_17;
END_VAR

  IF NOT Test_0.Finished AND NOT Test_0.FAILED THEN totalTests := totalTests + 1; Test_0(); END_IF;
  IF Test_0.Finished THEN testOutcomeArray[0] := TRUE; END_IF;
  IF NOT Test_1.Finished AND NOT Test_1.FAILED THEN totalTests := totalTests + 1; Test_1(); END_IF;
  IF Test_1.Finished THEN testOutcomeArray[1] := TRUE; END_IF;
  IF NOT Test_2.Finished AND NOT Test_2.FAILED THEN totalTests := totalTests + 1; Test_2(); END_IF;
  IF Test_2.Finished THEN testOutcomeArray[2] := TRUE; END_IF;
  IF NOT Test_3.Finished AND NOT Test_3.FAILED THEN totalTests := totalTests + 1; Test_3(); END_IF;
  IF Test_3.Finished THEN testOutcomeArray[3] := TRUE; END_IF;
  IF NOT Test_4.Finished AND NOT Test_4.FAILED THEN totalTests := totalTests + 1; Test_4(); END_IF;
  IF Test_4.Finished THEN testOutcomeArray[4] := TRUE; END_IF;
  IF NOT Test_5.Finished AND NOT Test_5.FAILED THEN totalTests := totalTests + 1; Test_5(); END_IF;
  IF Test_5.Finished THEN testOutcomeArray[5] := TRUE; END_IF;
  IF NOT Test_6.Finished AND NOT Test_6.FAILED THEN totalTests := totalTests + 1; Test_6(); END_IF;
  IF Test_6.Finished THEN testOutcomeArray[6] := TRUE; END_IF;
  IF NOT Test_7.Finished AND NOT Test_7.FAILED THEN totalTests := totalTests + 1; Test_7(); END_IF;
  IF Test_7.Finished THEN testOutcomeArray[7] := TRUE; END_IF;
  IF NOT Test_8.Finished AND NOT Test_8.FAILED THEN totalTests := totalTests + 1; Test_8(); END_IF;
  IF Test_8.Finished THEN testOutcomeArray[8] := TRUE; END_IF;
  IF NOT Test_9.Finished AND NOT Test_9.FAILED THEN totalTests := totalTests + 1; Test_9(); END_IF;
  IF Test_9.Finished THEN testOutcomeArray[9] := TRUE; END_IF;
  IF NOT Test_10.Finished AND NOT Test_10.FAILED THEN totalTests := totalTests + 1; Test_10(); END_IF;
  IF Test_10.Finished THEN testOutcomeArray[10] := TRUE; END_IF;
  IF NOT Test_11.Finished AND NOT Test_11.FAILED THEN totalTests := totalTests + 1; Test_11(); END_IF;
  IF Test_11.Finished THEN testOutcomeArray[11] := TRUE; END_IF;
  IF NOT Test_12.Finished AND NOT Test_12.FAILED THEN totalTests := totalTests + 1; Test_12(); END_IF;
  IF Test_12.Finished THEN testOutcomeArray[12] := TRUE; END_IF;
  IF NOT Test_13.Finished AND NOT Test_13.FAILED THEN totalTests := totalTests + 1; Test_13(); END_IF;
  IF Test_13.Finished THEN testOutcomeArray[13] := TRUE; END_IF;
  IF NOT Test_14.Finished AND NOT Test_14.FAILED THEN totalTests := totalTests + 1; Test_14(); END_IF;
  IF Test_14.Finished THEN testOutcomeArray[14] := TRUE; END_IF;
  IF NOT Test_15.Finished AND NOT Test_15.FAILED THEN totalTests := totalTests + 1; Test_15(); END_IF;
  IF Test_15.Finished THEN testOutcomeArray[15] := TRUE; END_IF;
  IF NOT Test_16.Finished AND NOT Test_16.FAILED THEN totalTests := totalTests + 1; Test_16(); END_IF;
  IF Test_16.Finished THEN testOutcomeArray[16] := TRUE; END_IF;
  IF NOT Test_17.Finished AND NOT Test_17.FAILED THEN totalTests := totalTests + 1; Test_17(); END_IF;
  IF Test_17.Finished THEN testOutcomeArray[17] := TRUE; END_IF;

  passedTests := 0;
  FOR i:=0 TO 17 DO
    IF testOutcomeArray[i]=TRUE THEN passedTests := passedTests+1; END_IF;
  END_FOR;
END_PROGRAM
